TYPE
    ST_HalfAuto_Storage :
    STRUCT
    END_STRUCT
END_TYPE

(* stored: Version 1.1.0.1, ProductVersion 3.1.4024.13
   DUT ST_HalfAuto_Storage: Id {b1d49c6e-8006-4836-ae82-5cec881b127a} *)
